// LS Electric XG5000 project: 8_21
// PLC LSPLC
// module base 0 slot 0: 입출력 모듈:XBC-DR14E (DC 24V 입력 8점, 릴레이 출력 6점)

PROGRAM NewProgram (task: 스캔 프로그램)

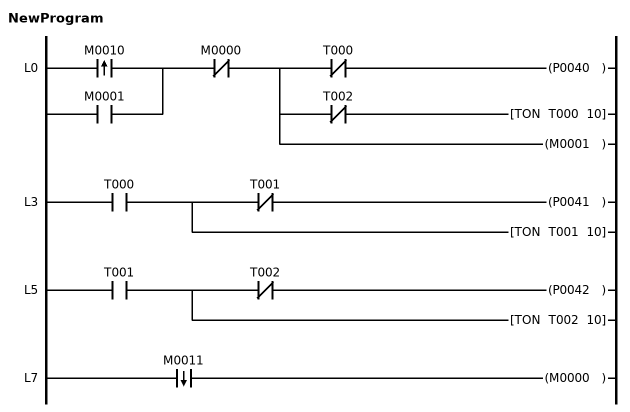
; L0
LOADP     M0010
OR        M0001
AND NOT   M0000
MPUSH
AND NOT   T000
OUT       P0040
MLOAD
AND NOT   T002
TON       T000 10
MPOP
OUT       M0001
; L3
LOAD      T000
MPUSH
AND NOT   T001
OUT       P0041
MPOP
TON       T001 10
; L5
LOAD      T001
MPUSH
AND NOT   T002
OUT       P0042
MPOP
TON       T002 10
; L7
LOADN     M0011
OUT       M0000